{attribute wpf [Container(Layout.Tabs)]}
PROGRAM MAIN
VAR
	{attribute wpf [Container(Layout.Stack)]}
	{attribute addProperty Name "Hello world"}
	Hello_World : STRING;
	{attribute addProperty Name "Counter"}
	Counter :INT;
	{attribute addProperty Name "Change me"}
	Variable :STRING;

//	{attribute wpf [Container(Layout.Stack)]}
//	_testStruct : stTestStruct;		
END_VAR

Hello_World := 'This is message from PLC!' ;
Counter := Counter +1 ;

END_PROGRAM

(* stored: Version 1.1.0.1, ProductVersion 3.1.4024.4
   POU MAIN: Id {2aec7386-fec2-4299-8c2e-88bb20ee3274}, SpecialFunc None *)
